// TIA Portal V20 export
TYPE "typeEm5MonitoringCmStatus"
// stored: Access Published, Namespace Unit1
   STRUCT
      NgManualInputAxis { ExternalWritable := 'False'} : "LBC_typeAxis64PosControlNodeMonitoring";
      MagazineAxis { ExternalWritable := 'False'} : "LBC_typeAxis64PosControlNodeMonitoring";
      ngManualInputCyl { ExternalWritable := 'False'} : "LBC_typeTwoWayActuatorControlNodeMonitoring";
      ngManualInputVac1 { ExternalWritable := 'False'} : "LBC_typeTwoWayActuatorControlNodeMonitoring";
      ngManualInputVac2 { ExternalWritable := 'False'} : "LBC_typeTwoWayActuatorControlNodeMonitoring";
      ngManualInputVib1 { ExternalWritable := 'False'} : "LBC_typeTwoWayActuatorControlNodeMonitoring";
      ngManualInputVib2 { ExternalWritable := 'False'} : "LBC_typeTwoWayActuatorControlNodeMonitoring";
      magazineLockCyl { ExternalWritable := 'False'} : "LBC_typeTwoWayActuatorControlNodeMonitoring";
      ngManualMagElectrodeDetectSen { ExternalWritable := 'False'} : "LBC_typeDigitalSignalControlNodeMonitoring";
      ngManualMagDetectSen { ExternalWritable := 'False'} : "LBC_typeDigitalSignalControlNodeMonitoring";
      ngManualMagFullSen { ExternalWritable := 'False'} : "LBC_typeDigitalSignalControlNodeMonitoring";
      ngManualElectrodeDetectSen { ExternalWritable := 'False'} : "LBC_typeDigitalSignalControlNodeMonitoring";
   END_STRUCT;
END_TYPE
